PROGRAM pouS3Alarms
VAR
	idbMsgAlarm: FB_CheckMessageBounds;

END_VAR

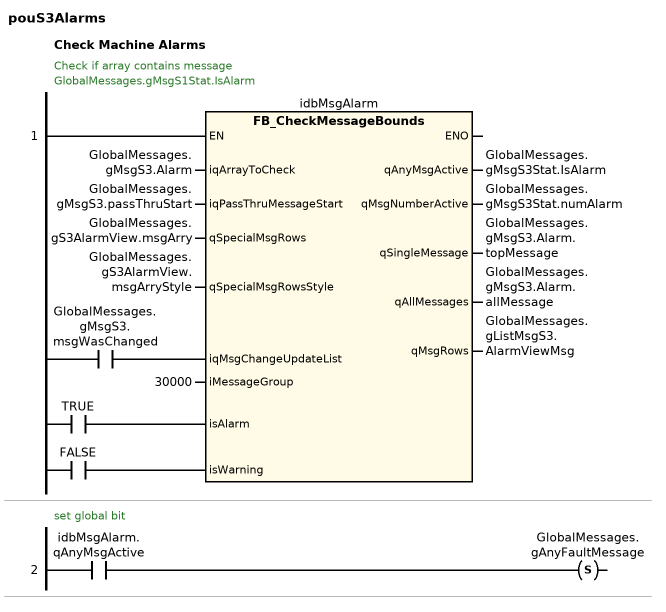
// NETWORK 1: Check Machine Alarms
// Check if array contains message
//
// GlobalMessages.gMsgS1Stat.IsAlarm
idbMsgAlarm(
    iqArrayToCheck := GlobalMessages.gMsgS3.Alarm,
    iqPassThruMessageStart := GlobalMessages.gMsgS3.passThruStart,
    qSpecialMsgRows := GlobalMessages.gS3AlarmView.msgArry,
    qSpecialMsgRowsStyle := GlobalMessages.gS3AlarmView.msgArryStyle,
    iqMsgChangeUpdateList := GlobalMessages.gMsgS3.msgWasChanged,
    iMessageGroup := 30000,
    isAlarm := TRUE,
    isWarning := FALSE,
    qAnyMsgActive => GlobalMessages.gMsgS3Stat.IsAlarm,
    qMsgNumberActive => GlobalMessages.gMsgS3Stat.numAlarm,
    qSingleMessage => GlobalMessages.gMsgS3.Alarm.topMessage,
    qAllMessages => GlobalMessages.gMsgS3.Alarm.allMessage,
    qMsgRows => GlobalMessages.gListMsgS3.AlarmViewMsg); // FB_CheckMessageBounds

// NETWORK 2
// set global bit
GlobalMessages.gAnyFaultMessage S= idbMsgAlarm.qAnyMsgActive;

END_PROGRAM

(* stored: Version 1.1.0.1, ProductVersion 3.1.4024.12
   POU pouS3Alarms: Id {7e55f54d-9cc6-45fd-9022-9e72fa8053a0}, SpecialFunc None *)
